# B&R Automation Studio project VisionSample (part 10)

#### Main.st - Init, cyclic, exit code
```iecst
// --------------------------------------------------------------------------------------------------------------------
// General vision task. This is a support task for the mappVision. The following functions are implemneted
// - Translate some values in text messages
// - Reset camera trigger when inspection is finsihed
// - Load vision application
// - Save diagnostic data
// Version 2.x (Check revision history for details)
// --------------------------------------------------------------------------------------------------------------------
PROGRAM _INIT

	FOR idx:= START_IDX TO NUM_CAMS BY 1 DO
		setupPointersAction;

		this.path := 'IF3.ST';
		tmpStr := USINT_TO_STRING(idx);
		brsstrcat(ADR(this.path),ADR(tmpStr));

		this.recipePVName := '::Vi_main:hmiInstance[';
		brsstrcat(ADR(this.recipePVName),ADR(tmpStr));
		brsstrcat(ADR(this.recipePVName),ADR('].in.recipe'));

		this.user.dataPvName := '::Vi_main:localInstance[';
		brsstrcat(ADR(this.user.dataPvName),ADR(tmpStr));
		brsstrcat(ADR(this.user.dataPvName),ADR('].user.data'));

		hmi.out.wsPort := 18000+idx*10;
		this.mappView.enable := TRUE;
		this.mappView.wsPort := hmi.out.wsPort;
		this.mappView.simulateConfig.activate := DiagCpuIsSimulated();
		this.mappView.simulateConfig.pFile := ADR('img');
		this.mappView.simulateConfig.useRandomNumbers := FALSE;
		this.mappView.simulateConfig.appendNumber := TRUE;
		this.mappView.simulateConfig.autoIncrementNumber := TRUE;
		this.mappView.simulateConfig.minNumber := 1;
		this.mappView.simulateConfig.maxNumber := 3;

		this.visionDiagFileDevice := 'VI_DIAG'; // File device is created in Files program (changes to USB if such is pluged in)

		hmi.out.camera.plNodeNr := idx;
		hmi.in.recipe.cam.focus := 200;
		hmi.in.recipe.cam.exposureTime := 100;

		hmi.in.cmd.resetInfo := TRUE;

		// -----------------------------------------------------------------------------------------------------------
		// Set camera specific data
		// -----------------------------------------------------------------------------------------------------------

		hmi.in.cmd.resultTabIndex := 5;
		CASE idx OF
			1:
				this.mappView.pMappLink := ADR(gCameraBlob);
				this.mappView.simulateConfig.pDevice := ADR('SIM_BLOB');
				hmi.out.camera.visionFunction := 'BLOB';
				hmi.out.usedVF.BLOB := TRUE;
				hmi.in.cmd.resultTabIndex := MIN(hmi.in.cmd.resultTabIndex,idx-1);
			2:
				this.mappView.pMappLink := ADR(gCameraCodeReading);
				this.mappView.simulateConfig.pDevice := ADR('SIM_CR');
				hmi.out.camera.visionFunction := 'Code Reader';
				hmi.out.usedVF.codeReader := TRUE;
				hmi.in.cmd.resultTabIndex := MIN(hmi.in.cmd.resultTabIndex,idx-1);
				(*hmi.out.VF.numResults*)
			3:
				this.mappView.pMappLink := ADR(gCameraMatch);
				this.mappView.simulateConfig.pDevice := ADR('SIM_MATCH');
				hmi.out.camera.visionFunction := 'Matching';
				hmi.out.usedVF.matching := TRUE;
				hmi.in.cmd.resultTabIndex := MIN(hmi.in.cmd.resultTabIndex,idx-1);
			4:
				this.mappView.pMappLink := ADR(gCameraMeasurement);
				this.mappView.simulateConfig.pDevice := ADR('SIM_MEAS');
				hmi.out.camera.visionFunction := 'Measurement';
				hmi.out.usedVF.measurement := TRUE;
				hmi.in.cmd.resultTabIndex := MIN(hmi.in.cmd.resultTabIndex,idx-1);
			5:
				this.mappView.pMappLink := ADR(gCameraOCR);
				this.mappView.simulateConfig.pDevice := ADR('SIM_OCR');
				hmi.out.camera.visionFunction := 'OCR';
				hmi.out.usedVF.OCR := TRUE;
				hmi.in.cmd.resultTabIndex := MIN(hmi.in.cmd.resultTabIndex,idx-1);
			6:
				this.mappView.pMappLink := ADR(gCameraPxl);
				this.mappView.simulateConfig.pDevice := ADR('SIM_PXCNT');
				hmi.out.camera.visionFunction := 'Pixel Counter';
				hmi.out.usedVF.pixelCounter := TRUE;
				hmi.in.cmd.resultTabIndex := MIN(hmi.in.cmd.resultTabIndex,idx-1);

		END_CASE

	END_FOR

END_PROGRAM

// -----------------------------------------------------------------------------------------------------------
// Cyclic part
// -----------------------------------------------------------------------------------------------------------
PROGRAM _CYCLIC

	FOR idx:= START_IDX TO NUM_CAMS BY 1 DO
		setupPointersAction;

		// -----------------------------------------------------------------------------------------------------------
		// Translate camera status in readable text
		// -----------------------------------------------------------------------------------------------------------
		brdkViBase_camStatusToString(hw.camera.in.status.cameraStatus,ADR(hmi.out.camera.statusText));

		// -----------------------------------------------------------------------------------------------------------
		// Check if vision cockpit is open
		// -----------------------------------------------------------------------------------------------------------
		hmi.out.camera.mappVisionActive := (hw.camera.in.status.cameraStatus AND 16#8000_0000) > 0;

		// -----------------------------------------------------------------------------------------------------------
		// Read camera hardware info
		// -----------------------------------------------------------------------------------------------------------

		IF hmi.in.cmd.resetInfo THEN
			hmi.in.cmd.resetInfo := FALSE;
			hmi.in.cameraInfo.distance := hmi.in.recipe.cam.focus;
			this.brdkViBase_getCameraInfo_0.execute := TRUE;
		END_IF

		this.brdkViBase_getCameraInfo_0.pDevicePath := ADR(this.path);
		this.brdkViBase_getCameraInfo_0.pInfo := ADR(hmi.in.cameraInfo);
		this.brdkViBase_getCameraInfo_0();

		IF hw.camera.out.par.focus <> hmi.in.recipe.cam.focus THEN
			hmi.in.cameraInfo.distance := hmi.in.recipe.cam.focus;
		END_IF

		IF hmi.in.cameraInfo.orderNr <> '' AND this.brdkViBase_getCameraInfo_0.status = ERR_OK THEN
			brdkViBase_calcOpticInfo(hmi.in.cameraInfo, hmi.out.camera.opticInfo); // calculate optic info based on defined info

			// set Camera flash options based on current camera
			hmi.out.camera.flashLightOptions[0] := '{"value":"0","text":"None"}';

			CASE hmi.in.cameraInfo.LED_color OF
				BRDKVIBASE_LED_COLOR_3_BLUE:
					hmi.out.camera.flashLightOptions[1] := '{"value":"3","text":"Blue"}';
				BRDKVIBASE_LED_COLOR_8_RED:
					hmi.out.camera.flashLightOptions[1] := '{"value":"1","text":"Red"}';
				BRDKVIBASE_LED_COLOR_A_UV:
					hmi.out.camera.flashLightOptions[1] := '{"value":"210","text":"Ultraviolet"}';
				BRDKVIBASE_LED_COLOR_D_IR:
					hmi.out.camera.flashLightOptions[1] := '{"value":"100","text":"Infrared"}';
				BRDKVIBASE_LED_COLOR_F_W:
					hmi.out.camera.flashLightOptions[1] := '{"value":"99","text":"White"}';
				BRDKVIBASE_LED_COLOR_Q_RGBL:
					hmi.out.camera.flashLightOptions[1] := '{"value":"1","text":"Red"}';
					hmi.out.camera.flashLightOptions[2] := '{"value":"2","text":"Green"}';
					hmi.out.camera.flashLightOptions[3] := '{"value":"3","text":"Blue"}';
					hmi.out.camera.flashLightOptions[4] := '{"value":"4","text":"Lime"}';

				BRDKVIBASE_LED_COLOR_R_RBIRW:
					hmi.out.camera.flashLightOptions[1] := '{"value":"1","text":"Red"}';
					hmi.out.camera.flashLightOptions[2] := '{"value":"3","text":"Blue"}';
					hmi.out.camera.flashLightOptions[3] := '{"value":"99","text":"White"}';
					hmi.out.camera.flashLightOptions[4] := '{"value":"100","text":"Infrared"}';
			END_CASE
		END_IF

		IF hw.io.in.nettime > this.axisTrig.nettimeLastCycle_us THEN
			this.axisTrig.powerlinkCycle_us	:= hw.io.in.nettime - this.axisTrig.nettimeLastCycle_us;
		ELSE
			this.axisTrig.powerlinkCycle_us	:= -2147483648-hw.io.in.nettime + 2147483647-this.axisTrig.nettimeLastCycle_us; // handle wrap around
		END_IF
		this.axisTrig.nettimeLastCycle_us	:= hw.io.in.nettime;

		// -----------------------------------------------------------------------------------------------------------
		// Image trigger (camera and lights)
		// -----------------------------------------------------------------------------------------------------------
		hmi.in.recipe.cam.flashColor := STRING_TO_USINT(hmi.in.recipe.cam.flashColorStr);
		hw.camera.out.par.focus 			:= hmi.in.recipe.cam.focus;
		hw.camera.out.par.flashSegment	 	:= hmi.in.recipe.cam.flashSegment;
		hw.camera.out.par.flashColor 		:= hmi.in.recipe.cam.flashColor;
		hw.camera.out.par.exposureTime 		:= hmi.in.recipe.cam.exposureTime;
		hw.camera.out.par.chromaticLock 	:= hmi.in.recipe.cam.chromaticLock;
		hw.camera.out.par.gainLevel 		:= hmi.in.recipe.cam.gainLevel;

		//-------------------------------------------------------------------------

		// Copy recipe data (e.g. enable, maximal number of results, etc.)
		hw.VF.blob.out			:=hmi.in.recipe.BLOB;
		hw.VF.codeReader.out	:= hmi.in.recipe.CR;
		hw.VF.matching.out		:=hmi.in.recipe.match;
		hw.VF.measurement.out	:=hmi.in.recipe.meassurement;
		hw.VF.ocr.out			:=hmi.in.recipe.OCR;
		hw.VF.pixelCnt.out		:=hmi.in.recipe.pxCnt;

		hmi.out.camera.processingTime:=hw.camera.in.status.cameraProcessingTime;

		CASE idx OF
			1:
				hmi.out.VF.processingTime := hw.VF.blob.in.common.functionProcessingTime;
				hmi.out.VF.numResults := hw.VF.blob.in.common.numResults;
			2:
				hmi.out.VF.processingTime := hw.VF.codeReader.in.common.functionProcessingTime;
				hmi.out.VF.numResults := hw.VF.codeReader.in.common.numResults;
			3:
				hmi.out.VF.processingTime := hw.VF.matching.in.common.functionProcessingTime;
				hmi.out.VF.numResults := hw.VF.matching.in.common.numResults;
			4:
				hmi.out.VF.processingTime := hw.VF.measurement.in.common.functionProcessingTime;
				hmi.out.VF.numResults := hw.VF.measurement.in.common.numResults;
			5:
				hmi.out.VF.processingTime := hw.VF.ocr.in.common.functionProcessingTime;
				hmi.out.VF.numResults := hw.VF.ocr.in.common.numResults;
			6:
				hmi.out.VF.processingTime := hw.VF.pixelCnt.in.common.functionProcessingTime;
				hmi.out.VF.numResults := hw.VF.pixelCnt.in.common.numResults;
		END_CASE;

		//-------------------------------------------------------------------------

		this.ioTrigger(CLK := hw.io.in.commonTrigger OR hw.io.in.individualTrigger);
		this.repetitiveTriggerTON.IN := hmi.in.recipe.repetitiveTrigger;
		this.repetitiveTriggerTON.PT := UDINT_TO_TIME(hmi.in.recipe.repetitiveTriggerInterval);
		this.repetitiveTriggerTON();

		// check if camera is ready for an image trigger and MappView have been updated
		IF this.brdkViBase_imgTrigger_0.ready AND NOT this.brdkViBase_imgTrigger_0.busy AND this.mappView.status = 0 THEN

			// Hmi manual trigger
			IF hmi.in.cmd.trigger OR this.repetitiveTriggerTON.Q THEN
				hmi.in.cmd.trigger 							:= FALSE;

				this.repetitiveTriggerTON(IN:=FALSE);

				this.brdkViBase_imgTrigger_0.trigger 		:= TRUE;
				this.brdkViBase_imgTrigger_0.delayNettime 	:= hw.io.in.nettime + gAxis.status.powerlinkCycleTime * 12+10000; // Calc nettime close to currnet time
				this.currentTriggerNum := 1;
			// Axis trigger
			ELSIF hmi.in.recipe.enableAxisTrigger AND
					gAxis.status.triggerTimeDelta >= (commonHmi.in.recipe.visionPreTriggerCycles * this.axisTrig.powerlinkCycle_us) AND
					gAxis.status.triggerTimeDelta <= ((commonHmi.in.recipe.visionPreTriggerCycles + 1) * this.axisTrig.powerlinkCycle_us) THEN

				this.brdkViBase_imgTrigger_0.trigger := TRUE;
				this.brdkViBase_imgTrigger_0.delayNettime := gAxis.status.nettime + gAxis.status.triggerTimeDelta; // Use time calculated in Axis program
			ELSIF hmi.in.recipe.enableIoTrigger AND this.ioTrigger.Q THEN

				this.brdkViBase_imgTrigger_0.trigger := TRUE;
				this.brdkViBase_imgTrigger_0.delayNettime := gAxis.status.nettime + hmi.in.recipe.ioTriggerDelay ; // Use time calculated in Axis program

			ELSIF this.currentTriggerNum < hmi.in.recipe.multiCaptureNum AND NOT hmi.in.recipe.repetitiveTrigger THEN

				this.brdkViBase_imgTrigger_0.trigger 		:= TRUE;
				this.brdkViBase_imgTrigger_0.delayNettime 	:= hw.io.in.nettime + gAxis.status.powerlinkCycleTime * 12+10000; // Calc nettime close to currnet time

				this.currentTriggerNum := 		this.currentTriggerNum +1;

			END_IF
		END_IF

		this.brdkViBase_imgTrigger_0.searchAcquisitonSettings := hmi.in.cmd.autoSearch;
		this.brdkViBase_imgTrigger_0.pCameraHw := ADR(hw.camera);
		this.brdkViBase_imgTrigger_0.numLights := NUM_LIGHTS;
		this.brdkViBase_imgTrigger_0.pLightHw := ADR(hw.lights);
		this.brdkViBase_imgTrigger_0.useCamColorForLight := hmi.in.recipe.useCamLedColorForLight;
		this.brdkViBase_imgTrigger_0.useCamExpTimeForLight := hmi.in.recipe.useCamExpTimeForLight;
		this.brdkViBase_imgTrigger_0.simulate.enable := DiagCpuIsSimulated();
		this.brdkViBase_imgTrigger_0.simulate.alwaysSimulateNonePresentLights := TRUE;
		this.brdkViBase_imgTrigger_0.simulate.imgProcessingDelay := T#300ms;
		this.brdkViBase_imgTrigger_0();

		// Manual Light trigger
		FOR i:=START_IDX TO NUM_LIGHTS BY 1 DO
			hmi.out.lights[i].plNodeNr := idx*16+UINT_TO_USINT(i-1);
			IF hmi.in.cmd.lights[i].flashTrigger THEN
				hw.lights[i].out.cmd.flashTrigger := TRUE;
				hw.lights[i].out.par.nettime := hw.io.in.nettime + gAxis.status.powerlinkCycleTime * commonHmi.in.recipe.visionPreTriggerCycles;
			END_IF

			IF 	hw.lights[i].out.cmd.flashTrigger AND hw.lights[i].out.par.nettime <= hw.io.in.nettime THEN
				hw.lights[i].out.cmd.flashTrigger := FALSE;
			END_IF
		END_FOR

		// -----------------------------------------------------------------------------------------------------------
		// New image ready and results
		// -----------------------------------------------------------------------------------------------------------
		// New image (hight for one scan)
		IF this.brdkViBase_imgTrigger_0.newImage THEN

			this.mappView.updateImage := NOT hmi.in.recipe.showOnlyLastImage OR this.currentTriggerNum = hmi.in.recipe.multiCaptureNum; // Trigger an update of the image on hmi
			this.DTGetTime_0(enable := TRUE);

			processResultsAction; // Process results action

		END_IF

		// -----------------------------------------------------------------------------------------------------------
		// Selection of specific result
		// -----------------------------------------------------------------------------------------------------------
		IF hmi.in.cmd.click THEN
			styleStringGeneration;
			hmi.in.cmd.click := FALSE;

			//VF
			brdkStrSubStr(ADR(tmpVF),ADR(hmi.in.cmd.elemId),1,1);
			//ID
			brsstrcpy(ADR(tmpID),ADR(hmi.in.cmd.elemId)+2);

			hmi.in.cmd.intElemId := STRING_TO_USINT(tmpID);
		END_IF

		IF hmi.in.cmd.intElemId <> this.oldIntElemID THEN
			this.oldIntElemID := hmi.in.cmd.intElemId;
			processResultsAction;
		END_IF

		// -----------------------------------------------------------------------------------------------------------
		// Auto search vision acquistion settings done (save found settings in recipe structure)
		// -----------------------------------------------------------------------------------------------------------

		// search Auto Focus done (hight for one scan)
		IF this.brdkViBase_imgTrigger_0.searchAcquisitonSettingsDone THEN
			hmi.in.cmd.autoSearch 			:= FALSE;
			hmi.in.recipe.cam.gainLevel 	:=	 hw.camera.in.status.gainLevel;
			hmi.in.recipe.cam.focus		 	:=	 hw.camera.in.status.focus;
			hmi.in.recipe.cam.exposureTime 	:=	 hw.camera.in.status.exposureTime;
			this.brdkViBase_imgTrigger_0.searchAcquisitonSettings := FALSE;
			hmi.in.cmd.trigger 				:= TRUE;
		END_IF

		// -----------------------------------------------------------------------------------------------------------
		// MappView get image to show om hmi
		// -----------------------------------------------------------------------------------------------------------

		IF DiagCpuIsSimulated() THEN
			this.mappView.imageFormat := BRDKVIIMG_IMG_TYPE_JPEG;
		ELSE
			this.mappView.imageFormat := commonHmi.in.recipe.imageFormat;
		END_IF
		this.mappView.jpegQuality := commonHmi.in.recipe.jpegQuality;
		this.mappView();

		// -----------------------------------------------------------------------------------------------------------
		// Save image to file devive F:/images
		// -----------------------------------------------------------------------------------------------------------
		CASE this.saveState OF
			0:

				IF (hmi.in.cmd.saveImage OR (this.mappView.newSvgReady AND commonHmi.in.recipe.saveAllImages))  AND gFiles.output.ready THEN
					hmi.in.cmd.saveImage := FALSE;

					// create filename with VF name and current date of the image
					brsstrcpy(ADR(this.tmpFileName),ADR(hmi.out.camera.visionFunction));
					brsstrcat(ADR(this.tmpFileName),ADR('-'));
					brdkViBase_dateTimeToString(this.DTGetTime_0.DT1,'%Y-%m-%d-%H-%M-%S',ADR(this.tmpFileName));

					brsstrcpy(ADR(this.brdkFileWrite.fileName),ADR(this.tmpFileName));

					CASE this.mappView.imageFormat OF
						BRDKVIIMG_IMG_TYPE_JPEG:
							brsstrcat(ADR(this.brdkFileWrite.fileName),ADR('.jpg'));
						BRDKVIIMG_IMG_TYPE_BMP:
							brsstrcat(ADR(this.brdkFileWrite.fileName),ADR('.bmp'));
					END_CASE

					this.brdkFileWrite.enable := TRUE;
					this.brdkFileWrite.dataLength := this.mappView.internal.getImage.destLen;
					this.brdkFileWrite.pData := this.mappView.internal.getImage.pDest;
					this.brdkFileWrite.overwrite := TRUE;
					this.brdkFileWrite.fileDevice := 'IMG';

					this.saveState := 10;
				END_IF
			10:

				IF this.brdkFileWrite.done THEN
					gFiles.input.refresh := TRUE;
					this.brdkFileWrite.enable := FALSE;
					this.saveState := 20;
				END_IF

			20:
				brsstrcpy(ADR(this.brdkFileWrite.fileName),ADR(this.tmpFileName));

				brsstrcat(ADR(this.brdkFileWrite.fileName),ADR('.svg'));
				this.brdkFileWrite.enable := TRUE;
				this.brdkFileWrite.dataLength := brsstrlen(ADR(hmi.out.svgOverlay));
				this.brdkFileWrite.pData := ADR(hmi.out.svgOverlay);
				this.brdkFileWrite.overwrite := TRUE;
				this.brdkFileWrite.fileDevice := 'IMG';

				this.saveState := 30;

			30:
				IF this.brdkFileWrite.done THEN
					gFiles.input.refresh := TRUE;
					this.brdkFileWrite.enable := FALSE;
					this.saveState := 0;
				END_IF

		END_CASE

		this.brdkFileWrite();

		// -----------------------------------------------------------------------------------------------------------
		// Save diagnostic data
		// -----------------------------------------------------------------------------------------------------------
		IF hmi.in.cmd.saveDiagnositc AND gFiles.output.ready THEN
			hmi.in.cmd.saveDiagnositc 			:= FALSE;

			// Delete old file first
			this.fileDelete.enable 					:= TRUE;
			this.fileDelete.pDevice 				:= ADR(this.visionDiagFileDevice);
			this.fileDelete.pName 					:= ADR(hmi.in.diagnosticFilename);

			// Upload diagnostic information
			this.viBaseSaveDiagData_0.MpLink 		:= this.mappView.pMappLink;
			this.viBaseSaveDiagData_0.DeviceName 	:= ADR(this.visionDiagFileDevice);
			this.viBaseSaveDiagData_0.FileName 		:= ADR(hmi.in.diagnosticFilename);
			hmi.out.camera.saveDiagStatus 			:= UINT_TO_DINT(ERR_FUB_BUSY);
		END_IF

		// file delete done or error (if file do not exsist)
		IF (this.fileDelete.enable AND this.fileDelete.status = ERR_OK) THEN
			this.fileDelete.enable 				:= FALSE;
			this.viBaseSaveDiagData_0.Execute 	:= TRUE;
		END_IF

		// Done
		IF (this.viBaseSaveDiagData_0.Done) THEN
			hmi.out.camera.saveDiagStatus		:= UINT_TO_DINT(ERR_OK);
			this.viBaseSaveDiagData_0.Execute 	:= FALSE;
		END_IF

		// Error
		IF (NOT this.viBaseSaveDiagData_0.Busy AND this.viBaseSaveDiagData_0.Error) THEN
			hmi.out.camera.saveDiagStatus		:= this.viBaseSaveDiagData_0.StatusID;
			this.viBaseSaveDiagData_0.Execute 	:= FALSE;
		END_IF

		this.viBaseSaveDiagData_0();
		this.fileDelete();

		// -----------------------------------------------------------------------------------------------------------
		// Get Vision application list from camera
		// -----------------------------------------------------------------------------------------------------------

		// trigger
		IF hmi.in.cmd.vaList.refresh THEN
			hmi.in.cmd.vaList.refresh 	:= FALSE;

			this.getVaList.Execute 		:= TRUE;
			this.getVaList.Format 		:= viBASE_FORMAT_PLAIN_TEXT;
			this.getVaList.List 		:= ADR(hmi.out.vaList.list);
			this.getVaList.ListLen 		:= SIZEOF(hmi.out.vaList.list);
			this.getVaList.MpLink 		:= this.mappView.pMappLink;
		END_IF

		// Done
		IF this.getVaList.Done THEN
			this.getVaList.Execute 		:= FALSE;
			hmi.out.vaList.length 		:= this.getVaList.NrEntries;
		END_IF

		// Error
		IF this.getVaList.Error THEN
			this.getVaList.Execute 		:= FALSE;
			hmi.out.vaList.lastError 	:= this.getVaList.StatusID;
		END_IF

		this.getVaList();

		// -----------------------------------------------------------------------------------------------------------
		// Load vision application
		// -----------------------------------------------------------------------------------------------------------

		// Trigger
		IF hmi.in.cmd.vaList.load AND brsstrlen(ADR(hmi.out.vaList.list[hmi.in.cmd.vaList.selectedIndex])) > 5 THEN
			hmi.in.cmd.vaList.load 						:= FALSE;

			this.viBaseLoadApplication_0.Execute 	:= TRUE;
			this.viBaseLoadApplication_0.MpLink		:= this.mappView.pMappLink;
			this.viBaseLoadApplication_0.Name		:= ADR(hmi.out.vaList.list[hmi.in.cmd.vaList.selectedIndex]);
			hmi.out.camera.vaLoad 					:= UINT_TO_DINT(ERR_FUB_BUSY);
		ELSE
			hmi.in.cmd.vaList.load := FALSE;
		END_IF

		// Done
		IF (this.viBaseLoadApplication_0.Done) THEN
			hmi.in.cmd.vaList.selectedIndex := 0;
			this.viBaseLoadApplication_0.Execute 	:= FALSE;
			hmi.out.camera.vaLoad 					:= UINT_TO_DINT(ERR_OK);
		END_IF

		// Error
		IF (NOT this.viBaseLoadApplication_0.Busy AND this.viBaseLoadApplication_0.Error) THEN
			this.viBaseLoadApplication_0.Execute 	:= FALSE;
			hmi.out.camera.vaLoad 					:= this.viBaseLoadApplication_0.StatusID;
		END_IF

		this.viBaseLoadApplication_0();

		// -----------------------------------------------------------------------------------------------------------
		// HMI stuff
		// -----------------------------------------------------------------------------------------------------------
		hmiAction;

		// -----------------------------------------------------------------------------------------------------------
		// Recipe handling (register recipse data structure
		// -----------------------------------------------------------------------------------------------------------
		this.mpRecipeRegVar.Enable 		:= gRecipe.out.active;
		this.mpRecipeRegVar.MpLink 		:= gRecipe.out.mpLink;
		this.mpRecipeRegVar.ConfirmSave := this.mpRecipeRegVar.SaveNotification;
		this.mpRecipeRegVar.Category 	:= ADR('Recipe');
		this.mpRecipeRegVar.PVName 		:= ADR(this.recipePVName);
		this.mpRecipeRegVar();

		// handle conversion from CR dropDown value to interger and back
		IF this.mpRecipeRegVar.UpdateNotification THEN
			hmi.in.recipe.CRTypeStr := USINT_TO_STRING(hmi.in.recipe.CR.symbolType);
		ELSE
			hmi.in.recipe.CR.symbolType := STRING_TO_USINT(hmi.in.recipe.CRTypeStr);
		END_IF

		this.user.mpRecipeRegVar.Enable 		:= gRecipe.out.active;
		this.user.mpRecipeRegVar.MpLink 	:= gRecipe.out.mpLink;
		this.user.mpRecipeRegVar.ConfirmSave := this.user.mpRecipeRegVar.SaveNotification;
		this.user.mpRecipeRegVar.Category 	:= ADR('Data');
		this.user.mpRecipeRegVar.PVName 	:= ADR(this.user.dataPvName);
		this.user.mpRecipeRegVar();

		// Clear ready for init (auto load) if data structures have not been registred
		IF NOT this.user.mpRecipeRegVar.Active OR NOT this.mpRecipeRegVar.Active THEN
			gRecipe.in.readyForInit := FALSE;
		END_IF

	END_FOR

	// -----------------------------------------------------------------------------------------------------------
	//Configure the pointers (this,hmi,hw etc.) show the correct data for that watch index
	// -----------------------------------------------------------------------------------------------------------
	watchIdx := LIMIT(START_IDX,watchIdx,NUM_CAMS);
	idx := watchIdx;
	setupPointersAction;

END_PROGRAM

PROGRAM _EXIT

	FOR idx:= START_IDX TO NUM_CAMS BY 1 DO
		setupPointersAction;

		this.mappView(enable := FALSE);
		this.mpRecipeRegVar(Enable := FALSE);
		this.user.mpRecipeRegVar(Enable := FALSE);
	END_FOR
END_PROGRAM
```

#### Types.typ
```iecst
TYPE
	local_axisTrig_typ : 	STRUCT
		nettimeLastCycle_us : DINT;
		powerlinkCycle_us : DINT;
		axisPositionNow : REAL;
		triggerPosDelta : REAL;
		triggerTimeDelta : DINT; (*In us*)
	END_STRUCT;
	local_vaList_typ : 	STRUCT
	END_STRUCT;
	local_typ : 	STRUCT
		path : STRING[100];
		brdkViBase_imgTrigger_0 : brdkViBase_imgTrigger;
		brdkViBase_getCameraInfo_0 : brdkViBase_getCameraInfo;
		mappView : {REDUND_UNREPLICABLE} brdkViImg_mappView;
		viBaseSaveDiagData_0 : ViBaseSaveDiagData;
		fileDelete : FileDelete;
		visionDiagFileDevice : STRING[10];
		viBaseLoadApplication_0 : ViBaseLoadApplication;
		axisTrig : local_axisTrig_typ;
		brdkFileWrite : brdkFileWrite;
		dtNow : DTStructure;
		DTGetTime_0 : DTGetTime;
		tmp2D : brdkViBase_2d_typ;
		strElemId : STRING[80];
		oldIntElemID : USINT;
		elemId : STRING[80];
		tmpAngle : LREAL;
		strStyle : STRING[240];
		mpRecipeRegVar : MpRecipeRegParSync;
		recipePVName : STRING[100];
		getVaList : ViBaseListApplication;
		tmpFileName : STRING[255];
		saveState : USINT;
		ioTrigger : R_TRIG;
		user : user_typ;
		currentTriggerNum : UINT;
		repetitiveTriggerTON : TON;
	END_STRUCT;
	hmi_typ : 	STRUCT
		in : hmi_in_typ;
		out : hmi_out_typ;
	END_STRUCT;
	hmi_out_vf_typ : 	STRUCT
		processingTime : UDINT;
		numResults : USINT;
		match : brdkViBase_hmi_match_in_typ;
		measurement : brdkViBase_hw_meas_in_typ;
		codeReader : brdkViBase_hmi_cr_in_typ;
		ocr : brdkViBase_hmi_OCR_in_typ;
		pixelCnt : brdkViBase_hmi_pxCnt_in_typ;
		blob : brdkViBase_hmi_blob_in_typ;
	END_STRUCT;
	hmi_out_lights_typ : 	STRUCT
		status : brdkViBase_light_hw_status_typ;
		common : brdkViBase_hw_in_common_typ;
		simulated : BOOL;
		connectedText : STRING[20];
		connected : BOOL;
		statusText : STRING[50];
		lightType : USINT;
		plNodeNr : USINT;
	END_STRUCT;
	hmi_out_camera_typ : 	STRUCT
		simulated : BOOL;
		connectedText : STRING[20];
		connected : BOOL;
		mappVisionActive : BOOL;
		processing : BOOL;
		ready : BOOL;
		statusText : STRING[50];
		plNodeNr : USINT;
		visionFunction : STRING[20];
		processingTime : UDINT;
		opticInfo : brdkViBase_opticInfo_typ;
		common : brdkViBase_hw_in_common_typ;
		hw : brdkViBase_cam_hw_in_status_typ;
		vaLoad : DINT;
		saveDiagStatus : DINT;
		flashLightOptions : ARRAY[0..4]OF STRING[100];
	END_STRUCT;
	hmi_out_vaList_typ : 	STRUCT
		list : ARRAY[0..99]OF ViBaseFormatPlainTextType;
		length : {REDUND_UNREPLICABLE} UINT;
		lastError : DINT;
	END_STRUCT;
	hmi_out_usedVF_typ : 	STRUCT
		pixelCounter : BOOL;
		measurement : BOOL;
		matching : BOOL;
		codeReader : BOOL;
		OCR : BOOL;
		BLOB : BOOL;
	END_STRUCT;
	hmi_out_typ : 	STRUCT
		svgOverlay : STRING[10000];
		wsPort : UINT;
		lights : ARRAY[START_IDX..NUM_LIGHTS]OF hmi_out_lights_typ;
		camera : hmi_out_camera_typ;
		VF : hmi_out_vf_typ;
		tableVF : hmi_out_vf_table_typ;
		vaList : hmi_out_vaList_typ;
		usedVF : hmi_out_usedVF_typ;
	END_STRUCT;
	hmi_in_cmd_flashSegment_typ : 	STRUCT
		top : BOOL := TRUE;
		bottom : BOOL := TRUE;
		right : BOOL := TRUE;
		left : BOOL := TRUE;
	END_STRUCT;
	hmi_in_cmd_vaList_typ : 	STRUCT
		refresh : BOOL;
		selectedIndex : UINT;
		load : BOOL;
	END_STRUCT;
	hmi_in_cmd_typ : 	STRUCT
		lights : ARRAY[START_IDX..NUM_LIGHTS]OF brdkViBase_light_hw_out_cmd_typ;
		flashSegment : hmi_in_cmd_flashSegment_typ;
		trigger : BOOL; (*Trigger a image*)
		autoSearch : BOOL; (*Start auto Search of exposure and focus for camra*)
		resetInfo : BOOL; (*Reset optic info to the current camera*)
		saveDiagnositc : BOOL; (*Save vision diagnostic *)
		saveImage : BOOL;
		intElemId : USINT := 1;
		elemId : STRING[80];
		click : BOOL;
		y : REAL;
		x : REAL;
		vaList : hmi_in_cmd_vaList_typ;
		resultTabIndex : USINT;
	END_STRUCT;
	hmi_in_recipe_draw_typ : 	STRUCT
		intShape : INT := 0; (*0 = None, 1=  rectangle, 2 = circle, 3 = triangle*)
		radius : REAL := 60;
		width : REAL := 80;
		length : REAL := 80;
		rotation : REAL := 0;
		fillColor : STRING[80] := ' fill: green;';
		activeStrokeColor : STRING[80] := ' stroke: orange;';
		strokeColor : STRING[80] := ' stroke: green;';
		strokeWidth : INT := 5;
		strokeOpac : REAL := 1;
		fillOpac : REAL := 0.3;
	END_STRUCT;
	hmi_in_typ : 	STRUCT
		cmd : hmi_in_cmd_typ;
		recipe : recipe_typ;
		cameraInfo : brdkViBase_camInfo_typ;
		diagnosticFilename : STRING[50];
		vaName : STRING[50];
		lightNum : USINT := 1;
	END_STRUCT;
	hw_io_in_typ : 	STRUCT
		nettime : DINT;
		commonTrigger : BOOL;
		individualTrigger : BOOL;
	END_STRUCT;
	hw_io_typ : 	STRUCT
		in : hw_io_in_typ;
	END_STRUCT;
	hw_typ : 	STRUCT
		camera : brdkViBase_cam_hw_typ;
		VF : hw_VF_typ;
		lights : ARRAY[START_IDX..NUM_LIGHTS]OF brdkViBase_light_hw_typ;
		io : hw_io_typ;
	END_STRUCT;
	hw_VF_typ : 	STRUCT
		codeReader : brdkViBase_hw_cr_10_typ;
		pixelCnt : brdkViBase_hw_pxCnt_10_typ;
		measurement : brdkViBase_hw_meas_10_typ;
		matching : brdkViBase_hw_match_10_typ;
		ocr : brdkViBase_hw_OCR_10_typ;
		blob : brdkViBase_hw_blob_10_typ;
	END_STRUCT;
	recipe_typ : 	STRUCT
		lights : ARRAY[START_IDX..NUM_LIGHTS]OF brdkViBase_light_hw_out_par_typ;
		cam : brdkViBase_cam_recipe_typ;
		BLOB : brdkViBase_hw_blob_out_typ;
		CR : brdkViBase_hw_cr_out_typ := (symbolType:=0);
		match : brdkViBase_hw_match_out_typ;
		meassurement : brdkViBase_hw_meas_out_typ;
		OCR : brdkViBase_hw_OCR_out_typ;
		pxCnt : brdkViBase_hw_pxCnt_out_typ;
		useCamExpTimeForLight : BOOL;
		useCamLedColorForLight : BOOL;
		ioTriggerDelay : DINT;
		enableIoTrigger : BOOL;
		multiCaptureNum : UINT := 1;
		showOnlyLastImage : BOOL;
		draw : hmi_in_recipe_draw_typ;
		enableAxisTrigger : BOOL;
		repetitiveTriggerInterval : UDINT;
		repetitiveTrigger : BOOL;
		CRTypeStr : STRING[20] := '0';
	END_STRUCT;
	common_hmi_in_cmd_typ : 	STRUCT
		deleteAllImage : BOOL;
		refreshVAlist : BOOL;
	END_STRUCT;
	common_hmi_in_typ : 	STRUCT
		recipe : common_recipe_typ;
		cmd : common_hmi_in_cmd_typ;
		dataFilePostName : STRING[255];
	END_STRUCT;
	common_hmi_typ : 	STRUCT
		in : common_hmi_in_typ;
	END_STRUCT;
	common_recipe_typ : 	STRUCT
		jpegQuality : USINT := 50;
		imageFormat : BRDKVIIMG_IMG_TYPE := BRDKVIIMG_IMG_TYPE_JPEG;
		visionPreTriggerCycles : DINT := 0;
		enableAxisTrigger : BOOL;
		saveAllImages : BOOL;
		saveSvg : BOOL;
		saveImage : BOOL;
	END_STRUCT;
	hmi_out_vf_table_cr_typ : 	STRUCT  (*Code reader structures*)
		BarcodeText : ARRAY[START_IDX..MAX_NUM_RESULTS]OF STRING[101];
		BarcodeType : ARRAY[START_IDX..MAX_NUM_RESULTS]OF USINT;
		PositionX : ARRAY[START_IDX..MAX_NUM_RESULTS]OF REAL;
		PositionY : ARRAY[START_IDX..MAX_NUM_RESULTS]OF REAL;
		Orientation : ARRAY[START_IDX..MAX_NUM_RESULTS]OF REAL;
		Grading : ARRAY[START_IDX..MAX_NUM_RESULTS]OF SINT;
	END_STRUCT;
	hmi_out_vf_table_blob_typ : 	STRUCT  (*Blob function structures*)
		ModelNumber : ARRAY[START_IDX..MAX_NUM_RESULTS]OF USINT;
		Clipped : ARRAY[START_IDX..MAX_NUM_RESULTS]OF BOOL;
		Area : ARRAY[START_IDX..MAX_NUM_RESULTS]OF REAL;
		PositionX : ARRAY[START_IDX..MAX_NUM_RESULTS]OF REAL;
		PositionY : ARRAY[START_IDX..MAX_NUM_RESULTS]OF REAL;
		Orientation : ARRAY[START_IDX..MAX_NUM_RESULTS]OF REAL;
		MeanGrayValue : ARRAY[START_IDX..MAX_NUM_RESULTS]OF USINT;
		Length : ARRAY[START_IDX..MAX_NUM_RESULTS]OF UDINT;
		Width : ARRAY[START_IDX..MAX_NUM_RESULTS]OF UDINT;
	END_STRUCT;
	hmi_out_vf_match_typ : 	STRUCT  (*Match function structures*)
		ModelNumber : ARRAY[START_IDX..MAX_NUM_RESULTS]OF USINT;
		Score : ARRAY[START_IDX..MAX_NUM_RESULTS]OF REAL;
		PositionX : ARRAY[START_IDX..MAX_NUM_RESULTS]OF REAL;
		PositionY : ARRAY[START_IDX..MAX_NUM_RESULTS]OF REAL;
		Orientation : ARRAY[START_IDX..MAX_NUM_RESULTS]OF REAL;
		Scale : ARRAY[START_IDX..MAX_NUM_RESULTS]OF REAL;
		RotCenterX : ARRAY[START_IDX..MAX_NUM_RESULTS]OF REAL;
		RotCenterY : ARRAY[START_IDX..MAX_NUM_RESULTS]OF REAL;
	END_STRUCT;
	hmi_out_vf_table_ocr_typ : 	STRUCT  (*OCR function structures*)
		Text : ARRAY[START_IDX..MAX_NUM_RESULTS]OF STRING[51];
		Grading : ARRAY[START_IDX..MAX_NUM_RESULTS]OF USINT;
		PositionX : ARRAY[START_IDX..MAX_NUM_RESULTS]OF REAL;
		PositionY : ARRAY[START_IDX..MAX_NUM_RESULTS]OF REAL;
		Orientation : ARRAY[START_IDX..MAX_NUM_RESULTS]OF REAL;
	END_STRUCT;
	hmi_out_vf_table_pxCnt_typ : 	STRUCT  (*OCR function structures*)
		ModelNumber : ARRAY[START_IDX..MAX_NUM_RESULTS]OF USINT;
		NumPixels : ARRAY[START_IDX..MAX_NUM_RESULTS]OF UDINT;
		MinGray : ARRAY[START_IDX..MAX_NUM_RESULTS]OF USINT;
		MaxGray : ARRAY[START_IDX..MAX_NUM_RESULTS]OF USINT;
		MeanGray : ARRAY[START_IDX..MAX_NUM_RESULTS]OF REAL;
		DeviationGray : ARRAY[START_IDX..MAX_NUM_RESULTS]OF REAL;
		MedianGray : ARRAY[START_IDX..MAX_NUM_RESULTS]OF USINT;
		ModelArea : ARRAY[START_IDX..MAX_NUM_RESULTS]OF UDINT;
		NumConnectedComponents : ARRAY[START_IDX..MAX_NUM_RESULTS]OF UINT;
		PositionX : ARRAY[START_IDX..MAX_NUM_RESULTS]OF REAL;
		PositionY : ARRAY[START_IDX..MAX_NUM_RESULTS]OF REAL;
	END_STRUCT;
	hmi_out_vf_table_meas_typ : 	STRUCT  (*MT function structures*)
		Result : ARRAY[START_IDX..MAX_NUM_RESULTS]OF DINT;
	END_STRUCT;
	hmi_out_vf_table_typ : 	STRUCT
		match : hmi_out_vf_match_typ;
		ocr : hmi_out_vf_table_ocr_typ;
		measurement : hmi_out_vf_table_meas_typ;
		pixelCnt : hmi_out_vf_table_pxCnt_typ;
		blob : hmi_out_vf_table_blob_typ;
		codeReader : hmi_out_vf_table_cr_typ;
	END_STRUCT;
END_TYPE
```

#### Variables1.var
```iecst
VAR CONSTANT
	START_IDX : USINT := 1;
END_VAR
VAR
	id : UDINT;
	tmpID : STRING[80];
	tmpVF : STRING[80];
	tmpStr : STRING[100];
	commonHmi : common_hmi_typ;
	p : USINT;
	tableNo : ARRAY[1..MAX_NUM_RESULTS] OF BYTE;
END_VAR
VAR CONSTANT
	MAX_NUM_RESULTS_M1 : USINT := MAX_NUM_RESULTS-1;
	MAX_NUM_RESULTS : USINT := 10;
	NUM_LIGHTS : USINT := 9;
END_VAR
VAR
	debug : BOOL;
END_VAR
VAR CONSTANT
	NUM_CAMS : USINT := 6;
END_VAR
VAR
	this : REFERENCE TO local_typ;
	hmi : REFERENCE TO hmi_typ;
	hw : REFERENCE TO hw_typ;
	hmiInstance : ARRAY[START_IDX..NUM_CAMS] OF hmi_typ;
	hwInstance : ARRAY[START_IDX..NUM_CAMS] OF hw_typ;
	localInstance : ARRAY[START_IDX..NUM_CAMS] OF local_typ;
	watchIdx : USINT;
	k : USINT;
	i : USINT;
	j : USINT;
	u : USINT;
	idx : USINT;
END_VAR
```

#### setupPointersAction.st
```iecst
ACTION setupPointersAction:

	hmi ACCESS ADR(hmiInstance[idx]);
	hw ACCESS ADR(hwInstance[idx]);
	this ACCESS ADR(localInstance[idx]);

END_ACTION
```

#### hmiAction.st
```iecst
ACTION hmiAction:

	IF DiagCpuIsSimulated() OR (NOT hw.camera.in.common.moduleOk AND this.brdkViBase_imgTrigger_0.simulate.alwaysSimulateNonePresentCamera) THEN
		hmi.out.camera.connected :=  TRUE;
		hmi.out.camera.simulated := TRUE;
	ELSE

		hmi.out.camera.simulated := FALSE;
		IF hw.camera.in.common.moduleOk THEN
			hmi.out.camera.connected :=  TRUE;
		ELSE
			hmi.out.camera.connected :=  FALSE;
		END_IF
	END_IF
	hmi.out.camera.processing := hw.camera.in.status.imageProcessingActive;
	hmi.out.camera.ready := this.brdkViBase_imgTrigger_0.ready AND NOT hmi.in.recipe.repetitiveTrigger;

	brsmemcpy(ADR(hmi.out.camera.hw),ADR(hw.camera.in.status),SIZEOF(hmi.out.camera.hw));
	brsmemcpy(ADR(hmi.out.camera.common),ADR(hw.camera.in.common),SIZEOF(hmi.out.camera.common));

	IF this.mpRecipeRegVar.UpdateNotification THEN

		hmi.in.cmd.flashSegment.top := hmi.in.recipe.cam.flashSegment.0;
		hmi.in.recipe.cam.flashSegment.1;
		hmi.in.cmd.flashSegment.left := 	hmi.in.recipe.cam.flashSegment.2;
		hmi.in.cmd.flashSegment.right := 	hmi.in.recipe.cam.flashSegment.3;

	ELSE
		hmi.in.recipe.cam.flashSegment.0 := hmi.in.cmd.flashSegment.top;
		hmi.in.recipe.cam.flashSegment.1 := hmi.in.cmd.flashSegment.bottom;
		hmi.in.recipe.cam.flashSegment.2 := hmi.in.cmd.flashSegment.left;
		hmi.in.recipe.cam.flashSegment.3 := hmi.in.cmd.flashSegment.right;
	END_IF

	FOR i:=START_IDX TO NUM_LIGHTS DO
		hmi.out.lights[i].common:=hw.lights[i].in.common;
		hmi.out.lights[i].status:=hw.lights[i].in.status;
		hw.lights[i].out.par.flashAngle:=hmi.in.recipe.lights[i].flashAngle;
		hw.lights[i].out.par.nettime:=this.brdkViBase_imgTrigger_0.delayNettime;

		IF hmi.in.recipe.useCamLedColorForLight THEN
			hw.lights[i].out.par.flashColor:=hmi.in.recipe.cam.flashColor;
		ELSE
			hw.lights[i].out.par.flashColor:=hmi.in.recipe.lights[i].flashColor;
		END_IF;

		IF hmi.in.recipe.useCamExpTimeForLight THEN
			hw.lights[i].out.par.exposureTime:=hmi.in.recipe.cam.exposureTime;
		ELSE
			hw.lights[i].out.par.exposureTime:=hmi.in.recipe.lights[i].exposureTime;
		END_IF;

	END_FOR;

	IF hmi.in.cmd.intElemId > 0 THEN

		IF hmi.in.cmd.intElemId <= hw.VF.blob.in.common.numResults THEN
			brdkViBase_blob_hw2hmi(hw.VF.blob.in.results[hmi.in.cmd.intElemId-1],hmi.out.VF.blob);
		END_IF

		IF hmi.in.cmd.intElemId <= hw.VF.codeReader.in.common.numResults THEN
			brdkViBase_cr_hw2hmi(hw.VF.codeReader.in.results[hmi.in.cmd.intElemId-1],hmi.out.VF.codeReader);
		END_IF

		IF hmi.in.cmd.intElemId <= hw.VF.matching.in.common.numResults THEN
			brdkViBase_match_hw2hmi(hw.VF.matching.in.results[hmi.in.cmd.intElemId-1],hmi.out.VF.match);
		END_IF

		IF hmi.in.cmd.intElemId <= hw.VF.measurement.in.common.numResults THEN
			brdkViBase_meas_hw2hmi(hw.VF.measurement.in.results[hmi.in.cmd.intElemId-1],hmi.out.VF.measurement);
		END_IF

		IF hmi.in.cmd.intElemId <= hw.VF.ocr.in.common.numResults THEN
			brdkViBase_ocr_hw2hmi(hw.VF.ocr.in.results[hmi.in.cmd.intElemId-1],hmi.out.VF.ocr);
		END_IF

		IF hmi.in.cmd.intElemId <= hw.VF.pixelCnt.in.common.numResults THEN
			brdkViBase_pxCnt_hw2hmi(hw.VF.pixelCnt.in.results[hmi.in.cmd.intElemId-1],hmi.out.VF.pixelCnt);
		END_IF
	ELSE
		// clear if 0
		brsmemset(ADR(hmi.out.VF.pixelCnt),0,SIZEOF(hmi.out.VF.pixelCnt));
		brsmemset(ADR(hmi.out.VF.ocr),0,SIZEOF(hmi.out.VF.ocr));
		brsmemset(ADR(hmi.out.VF.measurement),0,SIZEOF(hmi.out.VF.measurement));
		brsmemset(ADR(hmi.out.VF.match),0,SIZEOF(hmi.out.VF.match));
		brsmemset(ADR(hmi.out.VF.blob),0,SIZEOF(hmi.out.VF.blob));
		brsmemset(ADR(hmi.out.VF.codeReader),0,SIZEOF(hmi.out.VF.codeReader));
	END_IF

END_ACTION
```

#### processResultsAction.st
```iecst
ACTION processResultsAction:

	this.tmpAngle:= -(hmi.in.recipe.draw.rotation);

	// DRAW CIRCLES ON RESULTS
	hmi.out.svgOverlay := '';
	brsmemset(ADR(hmi.out.tableVF),0,SIZEOF(hmi.out.tableVF));

	//BLOB
	IF hw.VF.blob.in.common.numResults > 0 THEN
		FOR i:= 1 TO hw.VF.blob.in.common.numResults BY 1 DO

			//----------------------------------
			//          table results
			hmi.out.tableVF.blob.ModelNumber[i] := hw.VF.blob.in.results[i-1].modelNumber;
			hmi.out.tableVF.blob.Clipped[i] := hw.VF.blob.in.results[i-1].clipped;
			hmi.out.tableVF.blob.Area[i] := hw.VF.blob.in.results[i-1].area;
			hmi.out.tableVF.blob.PositionX[i] := DINT_TO_REAL(hw.VF.blob.in.results[i-1].positionX) /100.0;
			hmi.out.tableVF.blob.PositionY[i] :=  DINT_TO_REAL(hw.VF.blob.in.results[i-1].positionY) /100.0;
			hmi.out.tableVF.blob.Orientation[i] :=  DINT_TO_REAL(hw.VF.blob.in.results[i-1].orientation) /100.0;
			hmi.out.tableVF.blob.MeanGrayValue[i] := hw.VF.blob.in.results[i-1].meanGreyValue;
			hmi.out.tableVF.blob.Length[i] := hw.VF.blob.in.results[i-1].length;
			hmi.out.tableVF.blob.Width[i] := hw.VF.blob.in.results[i-1].width;

			//------------------------------------
			//			Overlay darwing
			this.tmp2D.x := DINT_TO_REAL(hw.VF.blob.in.results[i-1].positionX) / 100.0;
			this.tmp2D.y := DINT_TO_REAL(hw.VF.blob.in.results[i-1].positionY) / 100.0;
			this.tmpAngle:= -(hmi.out.tableVF.blob.PositionY[i]);
			// Style string generation
			// e.g.:'id="13" style="fill:blue;stroke:blue;stroke-width:5;fill-opacity:0.3;stroke-opacity:1"'
			this.strStyle := 'id="1';

			// Draw selested shape with specified parameters on the overlay
			styleStringGeneration;
		END_FOR;
	END_IF

	//CODE READER

	IF hw.VF.codeReader.in.common.numResults > 0 THEN
		FOR i:= 1 TO hw.VF.codeReader.in.common.numResults BY 1 DO

			//----------------------------------
			//          table results
			//Conversion of individual USINT values into strings for Code Reader
			brsmemcpy(ADR(hmi.out.tableVF.codeReader.BarcodeText[i]),ADR(hw.VF.codeReader.in.results[i-1].data),SIZEOF(hw.VF.codeReader.in.results[i-1].data));
			hmi.out.tableVF.codeReader.BarcodeType[i] 		:= hw.VF.codeReader.in.results[i-1].symbolType;
			hmi.out.tableVF.codeReader.Grading[i] 		:= hw.VF.codeReader.in.results[i-1].gradingValue;
			hmi.out.tableVF.codeReader.PositionX[i] 	:=  DINT_TO_REAL(hw.VF.codeReader.in.results[i-1].positionX) /100.0;
			hmi.out.tableVF.codeReader.PositionY[i] 	:=  DINT_TO_REAL(hw.VF.codeReader.in.results[i-1].positionY) /100.0;
			hmi.out.tableVF.codeReader.Orientation[i] 	:=  DINT_TO_REAL(hw.VF.codeReader.in.results[i-1].orientation) /100.0;

			//------------------------------------
			//			Overlay darwing

			this.tmp2D.x := DINT_TO_REAL(hw.VF.codeReader.in.results[i-1].positionX) / 100.0;
			this.tmp2D.y := DINT_TO_REAL(hw.VF.codeReader.in.results[i-1].positionY) / 100.0;
			this.tmpAngle:= -REAL_TO_LREAL(hmi.out.tableVF.codeReader.Orientation[i]);

			// Style string generation
			// e.g.:'id="13" style="fill:blue;stroke:blue;stroke-width:5;fill-opacity:0.3;stroke-opacity:1"'
			this.strStyle := 'id="2';

			styleStringGeneration;
		END_FOR;
	END_IF;

	//MATCHING

	IF hw.VF.matching.in.common.numResults > 0 THEN
		FOR i:= 1 TO hw.VF.matching.in.common.numResults BY 1 DO

			//----------------------------------
			//          table results
			hmi.out.tableVF.match.ModelNumber[i] := hw.VF.matching.in.results[i-1].modelNumber;
			hmi.out.tableVF.match.Score[i] :=  DINT_TO_REAL(hw.VF.matching.in.results[i-1].score) /100.0;
			hmi.out.tableVF.match.PositionX[i] :=  DINT_TO_REAL(hw.VF.matching.in.results[i-1].positionX) /100.0;
			hmi.out.tableVF.match.PositionY[i] :=  DINT_TO_REAL(hw.VF.matching.in.results[i-1].positionY) /100.0;
			hmi.out.tableVF.match.Orientation[i] :=  DINT_TO_REAL(hw.VF.matching.in.results[i-1].orientation) /100.0;
			hmi.out.tableVF.match.Scale[i] :=  DINT_TO_REAL(hw.VF.matching.in.results[i-1].scale) /100.0;

			//------------------------------------
			//			Overlay darwing

			this.tmp2D.x := DINT_TO_REAL(hw.VF.matching.in.results[i-1].positionX) / 100.0;
			this.tmp2D.y := DINT_TO_REAL(hw.VF.matching.in.results[i-1].positionY) / 100.0;
			this.tmpAngle:= -REAL_TO_LREAL(hmi.out.tableVF.blob.PositionY[i]);
			// Style string generation
			// e.g.:'id="13" style="fill:blue;stroke:blue;stroke-width:5;fill-opacity:0.3;stroke-opacity:1"'
			this.strStyle := 'id="3';

			// DRAW SELECTED SHAPE WITH SPECIFIED PARAMETERS ON THE OVERLAY
			styleStringGeneration;

		END_FOR;
	END_IF;

	//MEASUREMENT

	IF hw.VF.measurement.in.common.numResults > 0 THEN
		FOR i:=1 TO hw.VF.measurement.in.common.numResults DO
			hmi.out.tableVF.measurement.Result[i] := hw.VF.measurement.in.results[i-1].result;
		END_FOR;
	END_IF;

	//OCR

	IF hwInstance[5].VF.ocr.in.common.numResults > 0 THEN
		FOR i:= 1 TO hw.VF.ocr.in.common.numResults BY 1 DO
			//----------------------------------
			//          table results
			hmi.out.tableVF.ocr.Grading[i] := hw.VF.ocr.in.results[i-1].gradingValue;
			hmi.out.tableVF.ocr.PositionX[i] :=  DINT_TO_REAL(hw.VF.ocr.in.results[i-1].positionX) /100.0;
			hmi.out.tableVF.ocr.PositionY[i] :=  DINT_TO_REAL(hw.VF.ocr.in.results[i-1].positionY) /100.0;
			hmi.out.tableVF.ocr.Orientation[i] :=  DINT_TO_REAL(hw.VF.ocr.in.results[i-1].orientation) /100.0;
			//Conversion of individual USINT values into strings for OCR
			brsmemcpy(ADR(hmi.out.tableVF.ocr.Text[i]),ADR(hw.VF.ocr.in.results[i-1].data),SIZEOF(hw.VF.ocr.in.results[i-1].data));

			//------------------------------------
			//			Overlay darwing

			this.tmp2D.x := DINT_TO_REAL(hw.VF.ocr.in.results[i-1].positionX) / 100.0;
			this.tmp2D.y := DINT_TO_REAL(hw.VF.ocr.in.results[i-1].positionY) / 100.0;
			this.tmpAngle:= -REAL_TO_LREAL(hmi.out.tableVF.blob.PositionY[i]);
			// Style string generation
			// e.g.:'id="13" style="fill:blue;stroke:blue;stroke-width:5;fill-opacity:0.3;stroke-opacity:1"'

			this.strStyle := 'id="5';

			// DRAW SELECTED SHAPE WITH SPECIFIED PARAMETERS ON THE OVERLAY
			styleStringGeneration;

		END_FOR;
	END_IF;

	//PIXEL COUNT

	IF hwInstance[6].VF.pixelCnt.in.common.numResults > 0 THEN
		FOR i:= 1 TO hw.VF.pixelCnt.in.common.numResults BY 1 DO
			//----------------------------------
			//          table results
			hmi.out.tableVF.pixelCnt.ModelNumber[i] := hw.VF.pixelCnt.in.results[i-1].modelNumber;
			hmi.out.tableVF.pixelCnt.ModelArea[i] := hw.VF.pixelCnt.in.results[i-1].modelArea;
			hmi.out.tableVF.pixelCnt.NumPixels[i] := hw.VF.pixelCnt.in.results[i-1].numPixels;
			hmi.out.tableVF.pixelCnt.MinGray[i] := hw.VF.pixelCnt.in.results[i-1].minGray;
			hmi.out.tableVF.pixelCnt.MaxGray[i] := hw.VF.pixelCnt.in.results[i-1].maxGray;
			hmi.out.tableVF.pixelCnt.DeviationGray[i] :=  DINT_TO_REAL(hw.VF.pixelCnt.in.results[i-1].deviationGray) /100.0;
			hmi.out.tableVF.pixelCnt.MeanGray[i] :=  DINT_TO_REAL(hw.VF.pixelCnt.in.results[i-1].meanGray) /100.0;
			hmi.out.tableVF.pixelCnt.NumConnectedComponents[i] := hw.VF.pixelCnt.in.results[i-1].numConnectedComponents;
			hmi.out.tableVF.pixelCnt.PositionX[i] := DINT_TO_REAL(hw.VF.pixelCnt.in.results[i-1].positionX) /100.0;
			hmi.out.tableVF.pixelCnt.PositionY[i] := DINT_TO_REAL(hw.VF.pixelCnt.in.results[i-1].positionY) /100.0;

			//------------------------------------
			//			Overlay darwing

			this.tmp2D.x := DINT_TO_REAL(hw.VF.pixelCnt.in.results[i-1].positionX) / 100.0;
			this.tmp2D.y := DINT_TO_REAL(hw.VF.pixelCnt.in.results[i-1].positionY) / 100.0;
			this.tmpAngle := -REAL_TO_LREAL(hmi.in.recipe.draw.rotation);

			// Style string generation
			// e.g.:'id="13" style="fill:blue;stroke:blue;stroke-width:5;fill-opacity:0.3;stroke-opacity:1"'

			this.strStyle := 'id="6';

			styleStringGeneration;

		END_FOR;
	END_IF;

		END_ACTION
```

#### styleStringGeneration.st
```iecst
ACTION styleStringGeneration:

	IF hmi.in.recipe.draw.intShape > 0 THEN
		this.strElemId := UINT_TO_STRING(i);
		brsstrcat(ADR(this.strStyle),ADR(this.strElemId));					// string for element id attribute (value)
		brsstrcat(ADR(this.strStyle),ADR('" style="'));						// string for beginning of the style paramateres (text)
		brsstrcat(ADR(this.strStyle),ADR(hmi.in.recipe.draw.fillColor));		// string for fill color attribute (text + value)

		IF i = hmi.in.cmd.intElemId THEN
			brsstrcat(ADR(this.strStyle),ADR(hmi.in.recipe.draw.activeStrokeColor));
		ELSE
			brsstrcat(ADR(this.strStyle),ADR(hmi.in.recipe.draw.strokeColor));	// string for stroke color attribute (text + value)
		END_IF;

		brsstrcat(ADR(this.strStyle),ADR('stroke-width: ')); 				// string for stroke width attribute (text)
		tmpStr := INT_TO_STRING(hmi.in.recipe.draw.strokeWidth);
		brsstrcat(ADR(this.strStyle),ADR(tmpStr));	// string for stroke width attribute (value)
		brsstrcat(ADR(this.strStyle),ADR('; fill-opacity: ')); 				// string for fill opacity attribute (text)
		tmpStr := REAL_TO_STRING(hmi.in.recipe.draw.fillOpac);
		brsstrcat(ADR(this.strStyle),ADR(tmpStr)); 		// string for fill opacity attribute (value)
		brsstrcat(ADR(this.strStyle),ADR('; stroke-opacity: ')); 				// string for stroke opacity attribute (text)
		tmpStr := REAL_TO_STRING(hmi.in.recipe.draw.strokeOpac);
		brsstrcat(ADR(this.strStyle),ADR(tmpStr)); 	// string for stroke opacity attribute (value)
		brsstrcat(ADR(this.strStyle),ADR('"'));
	END_IF

	CASE hmi.in.recipe.draw.intShape OF
		0: // None

		1: // Rectangle
			brdkViGeom_drawSvgRectFromCP(this.tmp2D,hmi.in.recipe.draw.length,hmi.in.recipe.draw.width,this.tmpAngle,ADR(hmi.out.svgOverlay),ADR(this.strStyle));
		2: // Circle
			brdkViGeom_drawSvgCircle(this.tmp2D,hmi.in.recipe.draw.radius,ADR(hmi.out.svgOverlay),ADR(this.strStyle));
		3: // Triangle
			brdkViGeom_drawSvgTriFromCP(this.tmp2D,hmi.in.recipe.draw.length,hmi.in.recipe.draw.width,this.tmpAngle,ADR(hmi.out.svgOverlay),ADR(this.strStyle));
	END_CASE;

END_ACTION
```

#### user.typ
```iecst
TYPE
	user_stat_point_typ : 	STRUCT
		y : MTDataStatistics := (MovingWindowLength:=50,Update:=TRUE);
		x : MTDataStatistics := (MovingWindowLength:=50,Update:=TRUE);
	END_STRUCT;
	user_stat_typ : 	STRUCT
		distance : MTDataStatistics := (MovingWindowLength:=50,Update:=TRUE);
		point : ARRAY[0..1]OF user_stat_point_typ;
	END_STRUCT;
	user_points_typ : 	STRUCT
		p1 : brdkViBase_2d_typ;
		p2 : brdkViBase_2d_typ;
	END_STRUCT;
	user_typ : 	STRUCT
		p2 : brdkViBase_2d_typ;
		convert : LREAL;
		distanceMM : LREAL := 95;
		distance : LREAL;
		p1 : brdkViBase_2d_typ;
		statistic : user_stat_typ;
		currentPoints : user_points_typ;
		basePoints : user_points_typ;
		data : user_data_typ;
		mpRecipeRegVar : MpRecipeRegParSync;
		dataPvName : STRING[255];
	END_STRUCT;
	user_data_stat_typ : 	STRUCT
		var : REAL;
		std : REAL;
		data : ARRAY[0..49]OF LREAL;
		num : REAL;
		mean : REAL;
		max : REAL;
		min : {REDUND_UNREPLICABLE} REAL;
	END_STRUCT;
	user_data_typ : 	STRUCT
		distance : user_data_stat_typ;
		p2 : user_data_stat_point_typ;
		p1 : user_data_stat_point_typ;
	END_STRUCT;
	user_data_stat_point_typ : 	STRUCT
		x : user_data_stat_typ;
		y : user_data_stat_typ;
	END_STRUCT;
END_TYPE
```

### Package Logical/Programs/Recipe - Program to handle MpRecipe

### gRecipe.typ
```iecst
TYPE
	gRecipe_in_cmd_typ : 	STRUCT
		saveData : BOOL;
	END_STRUCT;
	gRecipe_in_typ : 	STRUCT
		cmd : gRecipe_in_cmd_typ;
		filename : STRING[255];
		readyForInit : BOOL;
	END_STRUCT;
	gRecipe_out_typ : 	STRUCT
		active : BOOL;
		mpLink : UDINT;
		init : BOOL;
	END_STRUCT;
	gRecipe_typ : 	STRUCT
		out : gRecipe_out_typ;
		in : gRecipe_in_typ;
	END_STRUCT;
END_TYPE
```

### gRecipe.var
```iecst
VAR
	gRecipe : gRecipe_typ;
END_VAR
```

### Program Logical/Programs/Recipe/Recipe (IEC)

#### Types.typ
```iecst
TYPE
	retain_typ : 	STRUCT
		lastLoadedName : STRING[255];
	END_STRUCT;
	local_typ : 	STRUCT
		mpRecipeUi : MpRecipeUI;
		mpRecipe : MpRecipeCsv;
		New_Member : USINT;
		delayTon : TON;
		autoLoadTon : TON;
	END_STRUCT;
	hmi_in_typ : 	STRUCT
		downloadDone : BOOL;
		download : BOOL;
	END_STRUCT;
	hmi_typ : 	STRUCT
		mpRecipe : MpRecipeUIConnectType;
		out : hmi_out_typ;
		in : hmi_in_typ;
	END_STRUCT;
	hmi_out_typ : 	STRUCT
		viewUrl : STRING[255];
		selectedName : STRING[255];
		downloadSrc : STRING[500];
		enableBtn : BOOL;
		lastLoaded : STRING[255];
	END_STRUCT;
END_TYPE
```

#### Variables.var
```iecst
VAR RETAIN
	retain : retain_typ;
END_VAR
VAR
	hmi : hmi_typ;
	this : local_typ;
END_VAR
```

#### Main.st
```iecst
PROGRAM _INIT
	(* Insert code here *)
	gRecipe.out.mpLink :=  ADR(gRecipeCsv_01);
	this.mpRecipe.DeviceName := ADR('RECIPE');
	this.mpRecipe.Category := ADR('Recipe');
	this.mpRecipe.MpLink := gRecipe.out.mpLink;

	this.mpRecipeUi.MpLink := gRecipe.out.mpLink;
	this.mpRecipeUi.UIConnect := ADR(hmi.mpRecipe);
	this.mpRecipeUi.UISetup.Confirmation.RecipeCreate 	:= FALSE;
	this.mpRecipeUi.UISetup.Confirmation.RecipeDelete 	:= FALSE;
	this.mpRecipeUi.UISetup.Confirmation.RecipeLoad 	:= FALSE;
	this.mpRecipeUi.UISetup.Confirmation.RecipeRename 	:= FALSE;
	this.mpRecipeUi.UISetup.Confirmation.RecipeSave 	:= FALSE;
	this.mpRecipeUi.UISetup.RecipeListScrollWindow		:= 5;
	this.mpRecipeUi.UISetup.RecipeListSize 				:= 10;

	IF  brsstrlen(ADR(retain.lastLoadedName)) > 0 THEN
		gRecipe.out.init := TRUE;
	END_IF

	this.autoLoadTon.PT := t#2s;
END_PROGRAM

PROGRAM _CYCLIC

	// if a data log should be saved instead (trigged from a program)
	IF gRecipe.in.cmd.saveData THEN
		gRecipe.in.cmd.saveData := FALSE;
		this.mpRecipe.DeviceName := ADR('DATA');
		this.mpRecipe.Category := ADR('Data');
		this.mpRecipe.FileName := ADR(gRecipe.in.filename);
		this.mpRecipe.Save := TRUE;
	END_IF

	// delay timer for auto load to ensure that all programs have run and had the chance to reset readyForInit if not ready
	this.autoLoadTon(IN := gRecipe.in.readyForInit);
	IF this.autoLoadTon.Q THEN
		this.mpRecipe.FileName 	:= ADR(retain.lastLoadedName);
		this.mpRecipe.Load 		:= TRUE;
		this.autoLoadTon.IN 	:= FALSE;
		gRecipe.out.init 		:= FALSE;
	END_IF

	// Set ready for init if init is needed. All programs will reset it they are not ready (reg var not done)
	gRecipe.in.readyForInit := gRecipe.out.init;

	this.mpRecipe(Enable 				:= gFiles.output.ready);
	this.mpRecipeUi(Enable 				:= this.mpRecipe.Active);
	gRecipe.out.active 					:= this.mpRecipe.Active;

	IF hmi.out.lastLoaded 	 <> this.mpRecipe.Info.LastLoadedRecipe AND brsstrcmp(this.mpRecipe.Category,ADR('Recipe')) = 0 THEN
		 hmi.out.lastLoaded	:= retain.lastLoadedName 	:= this.mpRecipe.Info.LastLoadedRecipe;
		this.mpRecipe.UpdateNotification := TRUE;
	ELSE
		this.mpRecipe.UpdateNotification := FALSE;
	END_IF

	IF hmi.mpRecipe.New.Create THEN
		hmi.out.lastLoaded	:= retain.lastLoadedName 	:= hmi.mpRecipe.New.FileName;
	END_IF

	hmi.out.selectedName 	:= hmi.mpRecipe.Recipe.List.Names[hmi.mpRecipe.Recipe.List.SelectedIndex];

	IF this.mpRecipe.CommandDone THEN
		this.mpRecipe.DeviceName := ADR('RECIPE');
		this.mpRecipe.Category := ADR('Recipe');
		this.mpRecipe.FileName := 0;
		this.mpRecipe.Save := FALSE;
	END_IF

	hmi.out.viewUrl := 'FileDevice:';
	brsstrcat(ADR(hmi.out.viewUrl),this.mpRecipe.DeviceName);
	brsstrcat(ADR(hmi.out.viewUrl),ADR('/'));
	brsstrcat(ADR(hmi.out.viewUrl),ADR(hmi.out.selectedName));

	// Handle download of recipe files (will crated an js code that is embedded in an paper widget (SVG) that automatically triggers a download of the file
	IF hmi.in.download THEN
		hmi.in.download 	:= FALSE;
		this.delayTon.IN 	:= TRUE;
		this.delayTon.PT 	:= T#400ms;

		hmi.out.downloadSrc := '<script>function onSvgLoad() {const link = document.createElement("a");link.href = "/FileDevice:';
		brsstrcat(ADR(hmi.out.downloadSrc),this.mpRecipe.DeviceName);
		brsstrcat(ADR(hmi.out.downloadSrc),ADR('/'));
		brsstrcat(ADR(hmi.out.downloadSrc),ADR(hmi.out.selectedName));
		brsstrcat(ADR(hmi.out.downloadSrc),ADR('";link.download="'));
		brsstrcat(ADR(hmi.out.downloadSrc),ADR(hmi.out.selectedName));
		brsstrcat(ADR(hmi.out.downloadSrc),ADR('";link.click();}; onSvgLoad(); </script>'));
	END_IF
	// reset the embedded JS such that when enter the page its not downloaded again.
	IF this.delayTon.Q THEN
		this.delayTon.IN := FALSE;
		hmi.out.downloadSrc := '';
	END_IF
	this.delayTon();

	hmi.out.enableBtn := brsstrlen(ADR(hmi.mpRecipe.Recipe.List.Names[0])) > 0;
END_PROGRAM

PROGRAM _EXIT
	this.mpRecipe(Enable 	:= FALSE);
	this.mpRecipeUi(Enable 	:= FALSE);
	gRecipe.out.active 		:= FALSE;
END_PROGRAM
```

- user.typ (reference to Logical/Programs/User/user.typ)

- userActions.st (reference to Logical/Programs/User/userActions.st)

### RecTypes.typ
```iecst
(*------------------------------------------------------------------------------------------------------------------------------------------------------------------------------------------------------------------------*)
(*Global enumerations*)

TYPE
	recSTATE :
		( (*Recipe management state machine*)
		REC_WAIT,
		REC_REG_NAME,
		REC_REG_VAR,
		REC_CREATE_DIR,
		REC_READ_DIR,
		REC_READ_DIR_1,
		REC_READ_DIR_2,
		REC_READ_DIR_3,
		REC_GEN_FILE_NAME,
		REC_LOAD_SAVE,
		REC_DELETE,
		REC_RENAME,
		REC_VIEW,
		REC_DOWNLOAD,
		REC_DOWNLOAD_1,
		REC_DOWNLOAD_2,
		REC_DOWNLOAD_3,
		REC_DOWNLOAD_4,
		REC_UPLOAD,
		REC_UPLOAD_1,
		REC_UPLOAD_2,
		REC_UPLOAD_3,
		REC_UPLOAD_4,
		REC_UPLOAD_5,
		REC_UPLOAD_6,
		REC_ERROR
		);
	recTYPE :
		(
		typeCSV,
		typeXML
		);
END_TYPE

(*------------------------------------------------------------------------------------------------------------------------------------------------------------------------------------------------------------------------*)
(*Global structure*)

TYPE
	recERR : 	STRUCT  (*Recipe management error structure*)
		Text : WSTRING[200]; (* Error text *)
		State : recSTATE; (* Error step *)
	END_STRUCT;
	recCMD : 	STRUCT  (*Recipe management command structure*)
		Init : BOOL := TRUE; (*Init recipes managment*)
		New : BOOL; (*Create new recipe*)
		Load : BOOL; (*Load recipe*)
		Save : BOOL; (*Save recipe*)
		View : BOOL; (*View recipe*)
		Rename : BOOL; (*Rename recipe*)
		Delete : BOOL; (*Delete recipe*)
		Download : BOOL; (*Download recipe*)
		Upload : BOOL; (*Upload recipe*)
		ErrorReset : BOOL; (*Reset pending errors*)
	END_STRUCT;
	recPAR : 	STRUCT  (*Recipe management parameter structure*)
		RecipeName : WSTRING[REC_NAME_LENGTH]; (*Recipe name*)
		RecipeNameNew : WSTRING[REC_NAME_LENGTH]; (*New recipe name*)
		RecipeID : STRING[REC_NAME_LENGTH]; (*File name of the recipe*)
		Initialized : BOOL; (*Indicates that recipe management was initialized*)
		VisuSlotID : USINT; (*ID for connected web connection*)
		VisuEnableCommand : BOOL;
	END_STRUCT;
	recDAT : 	STRUCT  (*Recipe management data structure*)
		RecipeNames : ARRAY[0..REC_REC_NUM]OF WSTRING[REC_NAME_LENGTH]; (*Recipe unicode names*)
		RecipeIDs : ARRAY[0..REC_REC_NUM]OF STRING[REC_NAME_LENGTH]; (*File name of the recipes*)
		RecipeNum : UINT; (*Number of recipes*)
	END_STRUCT;
	recVIS : 	STRUCT  (*Recipe management visualization structure*)
		RecipeNames : ARRAY[0..REC_REC_NUM]OF WSTRING[REC_VIS_LENGTH]; (*Recipe names as mappView data provider*)
		RecipeNum : UINT; (*Number of visible recipes*)
		RecipeFilter : WSTRING[REC_NAME_LENGTH]; (*Only show recipes that fit this pattern*)
		RecipeSelect : WSTRING[REC_NAME_LENGTH]; (*Select recipe in listbox after command new or rename*)
		DownloadFileUrl : STRING[REC_NAME_LENGTH]; (*URL used with recipe download*)
		UploadOverwriteRequest : BOOL; (*Show message box to overwrite file*)
		UploadOverwriteResponse : USINT; (*Response from message box overwrite file*)
		ReloadUpload : BOOL; (*Reload upload button*)
		RecipeDoubleClick : USINT; (*Track double click event*)
		ViewFilePath : STRING[REC_VIS_LENGTH]; (*Full path for viewing file*)
		ViewFile : BOOL; (*Trigger that opens the fly out window when viewing recipes*)
		ShowMessageBoxError : BOOL; (*Show message box on error*)
	END_STRUCT;
	recMAIN : 	STRUCT  (*Recipe management main structure*)
		CMD : recCMD; (* Command structure *)
		PAR : recPAR; (* Parameter structure *)
		DAT : recDAT; (*Data structure*)
		VIS : ARRAY[0..REC_MAX_CLIENTS_ID]OF recVIS; (*Visualization structure*)
		ERR : recERR; (* Error structure *)
		StatusText : WSTRING[100]; (*Shows the result of the last command*)
		StatusNo : DINT; (* Error number *)
	END_STRUCT;
END_TYPE
```

### Library Logical/Programs/mappRecipe/Recipe_01

#### RecipeVariables.var
```iecst
(*------------------------------------------------------------------------------------------------------------------------------------------------------------------------------------------------------------------------*)
(*Local constants*)
VAR CONSTANT
	OK : USINT := 0; (*Constant for status OK *)
	REC_DOES_NOT_EXIST : UINT := 65535; (*Constant for record does not exist*)
	YES : USINT := 1;
	NO : USINT := 2;
END_VAR
(*------------------------------------------------------------------------------------------------------------------------------------------------------------------------------------------------------------------------*)
(*Local Variables*)
VAR
	RECIPE : REFERENCE TO recMAIN; (*Local recipe structure*)
	DeviceName : STRING[80]; (*Device name where the recipes are stored*)
	RecipeIDs : ARRAY[0..REC_REC_NUM] OF BOOL; (*Used with unicode option, keeps tracks of the IDs used*)
	RecipeIndex : UINT; (*Current recipe index*)
	RecipeName : WSTRING[REC_NAME_LENGTH]; (*Local recipe name*)
	RecipeNameNew : WSTRING[REC_NAME_LENGTH]; (*Local recipe new name*)
	RecipeFullFileName : STRING[200]; (*Full recipe name*)
	RecipeFilterOld : ARRAY[0..REC_MAX_CLIENTS_ID] OF WSTRING[REC_NAME_LENGTH]; (*Track filter change *)
	RecipeNumOld : ARRAY[0..REC_MAX_CLIENTS_ID] OF UINT;
	rec_state : recSTATE := REC_WAIT; (*Main step index *)
	animation : USINT := 0; (*Animation for working status	*)
	VisuSlotID : USINT; (*Slot of the visualization that is current used*)
	idx : UINT; (*Index*)
	idy : UINT; (*Index*)
	has_oversized_items : BOOL; (*Indicates that at least one recipe name exceeds the maximum length*)
	tmpStr1 : STRING[200]; (*Temporary string variable *)
	tmpStr2 : STRING[200]; (*Temporary string variable *)
	tmpWStr1 : WSTRING[REC_VIS_LENGTH]; (*Temporary unicode string variable *)
	tmpWStr2 : WSTRING[REC_VIS_LENGTH]; (*Temporary unicode string variable *)
	lDirReadData : fiDIR_READ_EX_DATA; (*File information structure*)
	taskID : UDINT; (*Task ID*)
	taskGroup : USINT; (*Task Group*)
	taskStatus : UINT; (*Status of task information*)
	pvADR : UDINT; (*Adress of global variable structure*)
	pvLEN : UDINT; (*Lenght of global variable structure*)
	pvStatus : UINT; (*Status of global variable information*)
	pvCnt : UINT; (*Counter for variable registration*)
	MpRecipeDone : BOOL; (*Generic status done*)
	MpRecipeError : BOOL; (*Genereic status error*)
	MpRecipeStatusID : DINT; (*Generic error details*)
	DoubleClickRecipeName : ARRAY[0..REC_MAX_CLIENTS_ID] OF TON_10ms; (*Timer for double click detection*)
	response_header : httpResponseHeader_t; (*Response header for download*)
	response_header_data : STRING[300]; (*Response header data*)
	upload_delay : TON_10ms; (*Wait for upload data to finish*)
	download_timeout : TON_10ms; (*Timeout when download must finish*)
	upload_response : STRING[600]; (*Response for upload*)
	file_name_start : DINT; (*Start of file name in upload data*)
	file_name_len : DINT; (*Length of file name in upload data*)
	file_data_start : DINT; (*Start of data in upload data*)
	file_data_len : DINT; (*Length of data in upload data*)
	item_name : STRING[REC_NAME_LENGTH]; (*Recipe name in upload data*)
END_VAR
(*------------------------------------------------------------------------------------------------------------------------------------------------------------------------------------------------------------------------*)
(*Local function calls*)
VAR
	DInfo : DirInfo;
	DOpen : DirOpen;
	DRead : DirReadEx;
	DClose : DirClose;
	DCreate : DirCreate;
	FOpen : FileOpen;
	FCreate : FileCreate;
	FRead : FileReadEx;
	FWrite : FileWrite;
	FClose : FileClose;
	FDelete : FileDelete;
	FRename : FileRename;
	WebserviceDownload : httpService := (0);
	WebServiceUpload : httpService := (0);
	AsMemPartCreate_0 : AsMemPartCreate;
	AsMemPartAllocClear_0 : AsMemPartAllocClear;
	MpRecipeCsv_0 : MpRecipeCsv;
	MpRecipeXml_0 : MpRecipeXml;
	MpRecipeRegPar_0 : MpRecipeRegPar;
	MpRecipeRegPar_1 : ARRAY[1..REC_VAR_NUM] OF MpRecipeRegPar;
	MpComGetLink_0 : MpComGetLink;
END_VAR
(*------------------------------------------------------------------------------------------------------------------------------------------------------------------------------------------------------------------------*)
(*Error numbers*)
VAR CONSTANT
	ERR_REC_TOO_MANY_CLIENTS : DINT := 50010; (*More than 3 clients try to connect to recipe management*)
	ERR_REC_NAME_EMPTY : DINT := 50100; (*Recipe name is empty*)
	ERR_REC_NAME_EXISTS : DINT := 50101; (*Recipe name already exists*)
	ERR_REC_NAME_LOST : DINT := 50102; (*Recipe name was not found*)
	ERR_REC_NAME_LENGTH : DINT := 50103; (*One or more recipe names exceeds maximum length*)
	ERR_REC_DEV_NAME_EMPTY : DINT := 50110; (*Device name is empty*)
	ERR_REC_VAR_NAME_EMPTY : DINT := 50120; (*Variable name is empty*)
	ERR_REC_VAR_NAME_MISSING : DINT := 50121; (*Variable name is missing from unicode recipe file*)
	ERR_REC_NOT_INITIALIZED : DINT := 50130; (*Recipemanagement is not initialized*)
	ERR_REC_REC_NUM : DINT := 50140; (*Maximum number of recipes reached*)
	ERR_REC_TASK_NAME : DINT := 50150; (*Task name is incorrect*)
	ERR_REC_MPLINK : DINT := 50160; (*MpLink name is incorrect*)
	ERR_MEM_ALLOC : UINT := 50300; (*Memory allocation for file upload and download failed*)
	ERR_MEM_DOWNLOAD : UINT := 50310; (*Size of download file exceeds maximum*)
	ERR_TIMEOUT_DOWNLOAD : UINT := 50320; (*Download response timed out*)
	ERR_POS_NAME_UPLOAD : UINT := 50400; (*Can not find filename in upload response*)
	ERR_SIZE_NAME_UPLOAD : UINT := 50401; (*Can not determine end of filename in upload response*)
	ERR_LEN_NAME_UPLOAD : UINT := 50402; (*Filename is too long in upload response*)
	ERR_POS_DATA_UPLOAD : UINT := 50403; (*Can not find data in upload response*)
	ERR_SIZE_DATA_UPLOAD : UINT := 50404; (*Can not determine end of data in upload response*)
	ERR_MEM_UPLOAD : UINT := 50410; (*Size of upload file exceeds maximum size*)
	ERR_UNICODE_UPLOAD : UINT := 50420; (*Upload is not supported when unicode is used*)
END_VAR
```

#### LocalFunctions.fun
```iecst
FUNCTION CreateError : recSTATE
	VAR_INPUT
		RECIPE : REFERENCE TO recMAIN;
		No : DINT;
		Text : WSTRING[200];
		State : recSTATE;
	END_VAR
END_FUNCTION

FUNCTION CreateMessage : BOOL
	VAR_INPUT
		TargetString : UDINT;
		Text : UDINT;
		RecipeName : UDINT;
		VisuSlotID : USINT;
	END_VAR
	VAR
		VisuSlotIDStr : WSTRING[5];
		tmpWStr1 : WSTRING[200];
	END_VAR
END_FUNCTION

FUNCTION FindRecName : UINT
	VAR_INPUT
		RECIPE : REFERENCE TO recMAIN;
		RecipeName : WSTRING[REC_NAME_LENGTH];
	END_VAR
	VAR
		idx : UINT;
	END_VAR
END_FUNCTION

FUNCTION InsertRecName : UINT
	VAR_INPUT
		RECIPE : REFERENCE TO recMAIN;
		new_name : WSTRING[REC_NAME_LENGTH];
		new_id : STRING[REC_NAME_LENGTH];
	END_VAR
	VAR
		idx : INT;
		idy : INT;
		lSort : DINT;
		lValue : DINT;
		tmpSTR : STRING[REC_NAME_LENGTH];
	END_VAR
END_FUNCTION

FUNCTION RemoveRecName : BOOL
	VAR_INPUT
		RECIPE : REFERENCE TO recMAIN;
		RecipeIndex : UINT;
	END_VAR
END_FUNCTION

FUNCTION IsInstrW : BOOL
	VAR_INPUT
		string1 : UDINT;
		string2 : UDINT;
	END_VAR
	VAR
		idx : UDINT;
	END_VAR
END_FUNCTION

FUNCTION WorkingStatus : USINT
	VAR_INPUT
		RECIPE : REFERENCE TO recMAIN;
		str : UDINT;
		animation : USINT;
	END_VAR
END_FUNCTION

FUNCTION WString2DataProvider : BOOL
	VAR_INPUT
		SourceString : UDINT;
		TargetString : UDINT;
	END_VAR
END_FUNCTION

FUNCTION ReplaceString : BOOL
	VAR_INPUT
		dataSTR : UDINT;
		searchSTR : UDINT;
		replaceSTR : UDINT;
		first : BOOL;
	END_VAR
	VAR
		idx : UDINT;
	END_VAR
END_FUNCTION

FUNCTION FindInMem : DINT
	VAR_INPUT
		data1 : UDINT;
		len1 : UDINT;
		data2 : UDINT;
		len2 : UDINT;
		direction : BOOL;
	END_VAR
	VAR
		idx : UDINT;
	END_VAR
END_FUNCTION
```

#### Exit.st
```iecst
PROGRAM _EXIT
	// --------------------------------------------------------------------------------------------------------------------
	// Cyclic function calls
	MpRecipeRegPar_0(Enable := FALSE);
	FOR idx:=1 TO REC_VAR_NUM DO
		MpRecipeRegPar_1[idx](Enable := FALSE);
		IF(REC_VAR_LIST[idx] = '') THEN
			EXIT;
		END_IF
	END_FOR;
	MpRecipeCsv_0(Enable := FALSE);
	MpRecipeXml_0(Enable := FALSE);

END_PROGRAM
```

#### Init.st
```iecst
// --------------------------------------------------------------------------------------------------------------------
//	Function:	Recipe management with mappRecipe
//  Version:	0.8
//	Changed:	31.03.2022
// --------------------------------------------------------------------------------------------------------------------

PROGRAM _INIT
	// ----------------------------------------------------------------------------------------

	// ----------------------------------------------------------------------------------------
	// Dont change anything below this line
	// ----------------------------------------------------------------------------------------

	// ----------------------------------------------------------------------------------------
	// Make sure global variable structure and task name are correct
	taskStatus := ST_ident(ADR(REC_THIS_TASK), taskGroup, ADR(taskID));
	pvStatus := PV_xgetadr(ADR(REC_THIS_TASK), ADR(pvADR), ADR(pvLEN));
	// Connect global and local structure
	IF(pvStatus = 0) THEN
		RECIPE ACCESS pvADR;
		brsmemset(ADR(RECIPE.ERR), 0 , SIZEOF(RECIPE.ERR));
		RECIPE.PAR.Initialized := FALSE;
	END_IF

	// ----------------------------------------------------------------------------------------
	// Get mapp link information
	MpComGetLink_0.Enable := TRUE;
	MpComGetLink_0.ComponentName := ADR(REC_MPLINK);
	MpComGetLink_0();
	// Create error
	IF(MpComGetLink_0.Error) THEN
		rec_state := CreateError(ADR(RECIPE), ERR_REC_MPLINK, "mplink name is incorrect", rec_state);
	END_IF

	// ----------------------------------------------------------------------------------------
	// Allocate memory for file upload and download
	AsMemPartCreate_0.enable	:= TRUE;
	AsMemPartCreate_0.len		:= REC_UPLOAD_DOWNLOAD_SIZE;
	AsMemPartCreate_0();
	IF AsMemPartCreate_0.status <> 0 THEN
		rec_state := CreateError(ADR(RECIPE), ERR_MEM_ALLOC, "file upload and download memory alloc failed", rec_state);
	ELSE
		AsMemPartAllocClear_0.enable	:= TRUE;
		AsMemPartAllocClear_0.ident		:= AsMemPartCreate_0.ident;
		AsMemPartAllocClear_0.len		:= REC_UPLOAD_DOWNLOAD_SIZE;
		AsMemPartAllocClear_0();
		IF AsMemPartAllocClear_0.status <> 0 THEN
			rec_state := CreateError(ADR(RECIPE), ERR_MEM_ALLOC, "file upload and download memory clear failed", rec_state);
		END_IF
	END_IF

	// ----------------------------------------------------------------------------------------
	// Generate HTML messages for web upload
	upload_response	:= '<html><body><form action="/uploadA.html" name="form_upload" method="post" enctype="multipart/form-data" >
	<label for="file-upload" style="font-weight:bold;font-family: sans-serif;font-size:16px;padding:15px 50px;10px;10px;" class="custom-file-upload">Upload</label>
	<input type="file" id="file-upload" style="display:none;" onchange="form.submit()" name="file_selected" content-type="application/octet-stream" />
	</form><body></html> ';
	WebServiceUpload.pServiceName := ADR('uploadA.html');
END_PROGRAM
```

### Program Logical/Proxy/Vi_Proxy (IEC)

#### Main.st - Init, cyclic, exit code
```iecst
PROGRAM _INIT
	TcpForward_0.ServerPort := 8888;
	TcpForward_0.ConnectToPort := 8080 ; 			// Port used by Vision
	TcpForward_0.Enable := TRUE ;

END_PROGRAM

PROGRAM _CYCLIC
	ipSTR := '192.168.200.';
	brsitoa(visSelectedSensor, ADR(nodeSTR));
	brsstrcat(ADR(ipSTR), ADR(nodeSTR));
	TcpForward_0.ConnectToIp := ipSTR; 				//Vision camera IP ( Node 1 on powerlink network )
	TcpForward_0();

END_PROGRAM

PROGRAM _EXIT
	TcpForward_0.Enable := FALSE;
	TcpForward_0();

END_PROGRAM
```

#### Variables.var - Local variables
```iecst
VAR
	nodeSTR : STRING[80];
	ipSTR : STRING[80];
	TcpForward_0 : TcpForward;
END_VAR
```

Listed in the project but not available here: Logical/Global.typ, Logical/Global.var, Logical/Libraries/IecCheck/IecCheck.fun, Logical/Libraries/brdk/brdkSTR/brdkSTR.typ, Logical/Vision/Vi_main/setupPointersAction.st, Logical/Vision/Axis/Types.typ, Logical/Vision/Vi_Color/Types.typ, Logical/Vision/Vi_Optics/Types.typ, Logical/mappRecipe/RecTypes.typ, Logical/old/mappRecipe/Recipe_01/Init.st, Logical/old/mappRecipe/Recipe_01/Exit.st, Logical/old/mappRecipe/Recipe_01/RecipeVariables.var, Logical/old/mappRecipe/Recipe_01/LocalFunctions.fun, Logical/old/mappRecipe/Vi_image/Main.st, Logical/old/mappRecipe/Vi_image/Types.typ, Logical/old/mappRecipe/Vi_image/Actions.st, Logical/old/mappRecipe/Vi_image/ViDrawCrosshair.st, Logical/old/mappRecipe/Vi_image/ViCreateWebDirFile.st, Logical/Programs/Vision/Vision/setupPointersAction.st, Logical/Proxy/Vi_Proxy/Types.typ
